KUKA KRL program: MacroTmpReadMe.src

&ACCESS RVP
&COMMENT ReadMe File
DEF  MacroTmpReadMe ( )

; This file only exists as a directory placeholder file.

END
